FUNCTION_BLOCK FB_CartCtrlInSurgery EXTENDS FB_CartCtrlBase
VAR_INPUT
END_VAR
VAR_OUTPUT
END_VAR
VAR
END_VAR

// override this function in each exact controller
METHOD PROTECTED calcCmdJntPos : BOOL
VAR_IN_OUT CONSTANT
	// slave cart joint data
	i_slaveCart :FB_SlaveCart;
END_VAR
m_cmdJntPos := i_slaveCart.curJntPos;
END_METHOD

// override this function in each exact controller
// NOTICE: set joint control mode here, and do some initialization if needed
METHOD PUBLIC init : BOOL
VAR_IN_OUT CONSTANT
	i_slaveCart	:FB_SlaveCart;
END_VAR
VAR_IN_OUT 
	r_cartCtrlCmd :ST_SlaveArmCtrlCmds;
END_VAR
SUPER^.init(i_slaveCart,r_cartCtrlCmd);

// update commands to arm
copyCmds(r_cartCtrlCmd);
END_METHOD

END_FUNCTION_BLOCK

(* stored: Version 1.1.0.1, ProductVersion 3.1.4024.12
   POU FB_CartCtrlInSurgery: Id {370f14c6-9840-4a91-9e20-703802e8b3c3}, SpecialFunc None
   Method calcCmdJntPos: Id {3e9f002b-d35e-465a-8bf1-4822cd40807b}
   Method init: Id {1b8a6a5f-9b04-4cc6-b433-0c731d080f40} *)
